Staubli VAL3: getSizeItem.pgx

public program getSizeItem(string x_sName, num& x_nSize, num x_nType)
begin
  switch  x_nType
    case 0
      x_nSize=size(sml:box[x_sName].pPointRx)
    break
    case 1
      x_nSize=size(sml:box[x_sName].pToSafePt)
    break
    case 2
      x_nSize=size(sml:box[x_sName].jToHome)
    break
  endSwitch
end
